// TwinCAT 3 PLC project PLC
// ProgramVersion: 3.1.4026.26
// libraries:
//   Tc2_Standard, * (Beckhoff Automation GmbH)
//   Tc2_System, * (Beckhoff Automation GmbH)
//   Tc2_Utilities, * (Beckhoff Automation GmbH)
//   Tc3_Database, * (Beckhoff Automation GmbH)
//   Tc3_EventLogger, * (Beckhoff Automation GmbH)
// project tree:
//   10_Generator/DUTs/ ST_GeneratorHmi.TcDUT
//   10_Generator/ITFs/ I_Generator.TcIO
//   10_Generator/POUs/ FB_Generator.TcPOU
//   20_RoomTemp/DUTs/ E_CoolingControlState.TcDUT, ST_CoolingControlHmi.TcDUT, ST_RoomTempHmi.TcDUT
//   20_RoomTemp/ITFs/ I_RoomTemp.TcIO
//   20_RoomTemp/POUs/ FB_CoolingControl.TcPOU, FB_RoomTemp.TcPOU, FB_RoomTempControl.TcPOU
//   40_Data/DUTs/ ST_Process_1_Measurements.TcDUT
//   40_Data/POUs/ FB_DataLogger.TcPOU, FB_PLC_DB_Mode.TcPOU, FB_SQL_DB_Mode.TcPOU
//   50_Library/Motors/ITFs/DUTs/ ST_ControlWord.TcDUT, ST_StatusWord.TcDUT
//   50_Library/Motors/ITFs/ I_Motor.TcIO
//   50_Library/Motors/POUs/ FB_MotorAbb.TcPOU, FB_MotorAbb_1.TcPOU
//   99_ESIMERKKI/DUTs/ ST_Esimerkki.TcDUT, ST_EsimerkkiHMI.TcDUT
//   99_ESIMERKKI/POUs/ FB_EsimerkkiToiminto.TcPOU
//   DUTs/ PriceItem.TcDUT, ST_Motors.TcDUT
//   GVLs/ GVL.TcGVL, Motors.TcGVL, Safety.TcGVL
//   / PlcTask.TcTTO
//   POUs/10_aika_ennen_meitä/ FB_AIKA.TcPOU (not stored), FB_HINNAN_ARPOMINEN.TcPOU (not stored), FB_RANK_PRICES.TcPOU
//   POUs/ MAIN.TcPOU
// real-time tasks:
//   TASK PlcTask: cycle T#10ms, priority 20, ADS port 350
// I/O:
//   DEVICE Device 1 (EtherCAT), AmsNetId 192.168.0.154.2.1
//     moottori (FECA-01) [ABB FECA-01 EtherCAT adapter]
// variable links:
//   PLC/PLC Instance <-> Device 1 (EtherCAT)/moottori (FECA-01)
//     PlcTask Inputs/Motors.coolingMotor.nSpeedActual <-> TxPDO 6 map/vl velocity actual value
//     PlcTask Inputs/Motors.coolingMotor.wStatusWord <-> TxPDO 6 map/Statusword
//     PlcTask Outputs/Motors.coolingMotor.nSpeedRef <-> RxPDO 6 map/vl target velocity
//     PlcTask Outputs/Motors.coolingMotor.wControlWord <-> RxPDO 6 map/Controlword

CONFIGURATION PLC
    RESOURCE PLC ON TwinCAT3
        TASK PlcTask(INTERVAL := T#10ms, PRIORITY := 20);
        PROGRAM MAIN WITH PlcTask : MAIN;
    END_RESOURCE
END_CONFIGURATION

// ---- 10_Generator/DUTs/ST_GeneratorHmi.TcDUT
TYPE ST_GeneratorHmi :
STRUCT
	bStart			: BOOL;
	bStop			: BOOL;
	bAltaanTaso		: INT;
	nSahkonKulutus	: INT;
END_STRUCT
END_TYPE

// ---- 20_RoomTemp/DUTs/E_CoolingControlState.TcDUT
{attribute 'qualified_only'}
{attribute 'strict'}
{attribute 'to_string'}
TYPE E_CoolingControlState :
(
	Auto := 0,
	Manual := 1,
	Stop	:= 2,
	Error	:= 3
);
END_TYPE

// ---- 20_RoomTemp/DUTs/ST_CoolingControlHmi.TcDUT
TYPE ST_CoolingControlHmi :
STRUCT
	// HMI -> PLC
	sName					: STRING;
	paramRoomTempSet		: REAL; //
	param_P					: REAL;	//--- PID säätimen parametrit hmi:ltä
	param_I					: REAL;	//
	Param_D					: REAL;	//
	
	bAuto					: BOOL; // Automaatti tila hmi:ltä
	nMotorManualSpeed		: INT;	// Manuaaliajon nopeus hmi:ltä
END_STRUCT
END_TYPE

// ---- 20_RoomTemp/DUTs/ST_RoomTempHmi.TcDUT
TYPE ST_RoomTempHmi :
STRUCT
	// PLC -> HMI
	nRoomTemperature		: REAL;
	sName					: STRING;
	
	// HMI -> PLC
	nValue					: INT := 5; // skaalaus HMI:ltä
	
END_STRUCT
END_TYPE

// ---- 40_Data/DUTs/ST_Process_1_Measurements.TcDUT
TYPE ST_Process_1_Measurements :
STRUCT
	//nID:			LINT;
	//tTime:		DATE_AND_TIME;
	sName:			STRING(50);
	fTemperature:	LREAL;
	fPressure:		LREAL;
	fFlowRate:		LREAL;
END_STRUCT
END_TYPE

// ---- 50_Library/Motors/ITFs/DUTs/ST_ControlWord.TcDUT
TYPE ST_ControlWord :
STRUCT
    // Bitti 0-3: Tilakone ohjaus
    SwitchOn            : BIT;  // Bit 0
    EnableVoltage       : BIT;  // Bit 1
    QuickStop           : BIT;  // Bit 2 — 0 = quick stop aktivoitu
    EnableOperation     : BIT;  // Bit 3

    // Bitti 4-6: Operaatiomoodi spesifinen
    OperationMode0      : BIT;  // Bit 4
    OperationMode1      : BIT;  // Bit 5
    OperationMode2      : BIT;  // Bit 6

    // Bitti 7: Vikareset
    FaultReset          : BIT;  // Bit 7 — nouseva reuna resetoi vian

    // Bitti 8: Halt
    Halt                : BIT;  // Bit 8 — 1 = pysäytä

    // Bitti 9-15: Valmistaja spesifinen
    Reserved9           : BIT;
    Reserved10          : BIT;
    Reserved11          : BIT;
    Reserved12          : BIT;
    Reserved13          : BIT;
    Reserved14          : BIT;
    Reserved15          : BIT;
END_STRUCT
END_TYPE

// ---- 50_Library/Motors/ITFs/DUTs/ST_StatusWord.TcDUT
TYPE ST_StatusWord :
STRUCT
    // Bitti 0-7: Tilakone status
    ReadyToSwitchOn     : BIT;  // Bit 0
    SwitchedOn          : BIT;  // Bit 1
    OperationEnabled    : BIT;  // Bit 2
    Fault               : BIT;  // Bit 3
    VoltageEnabled      : BIT;  // Bit 4
    QuickStop           : BIT;  // Bit 5 — 0 = quick stop aktivoitu
    SwitchOnDisabled    : BIT;  // Bit 6
    Warning             : BIT;  // Bit 7

    // Bitti 8-15
    ManufacturerSpec    : BIT;  // Bit 8
    Remote              : BIT;  // Bit 9  — 1 = väylä ohjaa
    TargetReached       : BIT;  // Bit 10 — 1 = tavoite saavutettu
    InternalLimitActive : BIT;  // Bit 11
    OpModeSpecific0     : BIT;  // Bit 12
    OpModeSpecific1     : BIT;  // Bit 13
    Reserved14          : BIT;  // Bit 14
    Reserved15          : BIT;  // Bit 15
END_STRUCT
END_TYPE

// ---- 99_ESIMERKKI/DUTs/ST_Esimerkki.TcDUT
TYPE ST_Esimerkki :
STRUCT
	
	// Tähän structiin kerätään kaikki Esimerkkitoiminnot, jos niitä on useampia. Helpottaa HMI toimintoja.
	
	stEsimerkki_1			: ST_EsimerkkiHMI;
	stEsimerkki_2			: ST_EsimerkkiHMI;
END_STRUCT
END_TYPE

// ---- 99_ESIMERKKI/DUTs/ST_EsimerkkiHMI.TcDUT
TYPE ST_EsimerkkiHMI :
STRUCT
	bTieto1		: BOOL;
	bTieto2		: BOOL;
	nArvo1		: INT;
END_STRUCT
END_TYPE

// ---- DUTs/PriceItem.TcDUT

TYPE PriceItem : 
STRUCT 
	price : REAL;
	index : INT; 
END_STRUCT 
END_TYPE

// ---- DUTs/ST_Motors.TcDUT
TYPE ST_Motors :
STRUCT
	sName			: STRING;
	bAuto			: BOOL;
	bManual			: BOOL;
	bStop			: BOOL;
	bManualFw		: BOOL;
	bManualBw		: BOOL;
	nManualSpeed	: REAL := 20.0;
	bReset			: BOOL;
	
END_STRUCT
END_TYPE

// ---- GVLs/GVL.TcGVL
{attribute 'qualified_only'}
VAR_GLOBAL
	nTime_multiplier:		INT:=1;
	nSeconds:				INT;
	nMinutes:				INT;
	nHours:					INT;
	nCycle:					INT;
	nMontakohalvinta:		INT(1..95):=20;
	nMontakokalleinta:		INT(1..95):=20;
	nHintaRajaPumppaus:		REAL :=3.0;
	nHintaRajaTuotanto:		REAL :=7.0;
	fprice:					REAL;
	
	// DUT:eissa määriteltiin mitä tietoja structit sisältää. Tässä tehdään muuttuja structissa, jossa tieto asuu. yhdistetään HMI:hin
	stEsimerkki				: ST_Esimerkki;
	
	stGenerator				: ST_GeneratorHmi;
	// Laitoin genun GVL:ään -> helppo työntää rajapinnan kautta tietoja esim roomtempille.
	fbGenerator				: FB_Generator;
	
	stRoomTemp				: ST_RoomTempHmi;
	fbRoomtemp				: FB_RoomTemp;
	
	stCoolingControl		: ST_CoolingControlHmi;
	
	fbDataLogger			: FB_DataLogger;
END_VAR

// ---- GVLs/Motors.TcGVL
{attribute 'qualified_only'}
VAR_GLOBAL
	
	stMotors		: ST_Motors;
	
	
	// Motors
    {attribute 'TcLinkTo' := '.wControlWord := TIID^Device 1 (EtherCAT)^moottori (FECA-01)^RxPDO 6 map^Controlword;
                              .wStatusWord 	:= TIID^Device 1 (EtherCAT)^moottori (FECA-01)^TxPDO 6 map^Statusword;
							  .nSpeedRef	:= TIID^Device 1 (EtherCAT)^moottori (FECA-01)^RxPDO 6 map^vl target velocity;
							  .nSpeedActual := TIID^Device 1 (EtherCAT)^moottori (FECA-01)^TxPDO 6 map^vl velocity actual value'}	
	coolingMotor		: FB_MotorAbb;
END_VAR

// ---- GVLs/Safety.TcGVL
{attribute 'qualified_only'}
VAR_GLOBAL
END_VAR

// ---- 10_Generator/ITFs/I_Generator.TcIO
INTERFACE I_Generator

PROPERTY bRunning : BOOL
GET
END_GET
END_PROPERTY

PROPERTY nHeat : REAL
GET
END_GET
SET
END_SET
END_PROPERTY

END_INTERFACE

// ---- 20_RoomTemp/ITFs/I_RoomTemp.TcIO
INTERFACE I_RoomTemp

PROPERTY nRoomTemp : REAL
GET
END_GET
END_PROPERTY

END_INTERFACE

// ---- 50_Library/Motors/ITFs/I_Motor.TcIO
INTERFACE I_Motor

PROPERTY bAuto : BOOL
GET
END_GET
SET
END_SET
END_PROPERTY

PROPERTY bEnable : BOOL
GET
END_GET
SET
END_SET
END_PROPERTY

PROPERTY bRunning : BOOL
GET
END_GET
END_PROPERTY

PROPERTY nSpeed : INT
GET
END_GET
SET
END_SET
END_PROPERTY

END_INTERFACE

// ---- POUs/MAIN.TcPOU
PROGRAM MAIN
VAR
	// ESIMERKKI TOIMINTO
	fbEsimerkkiToiminto		: FB_EsimerkkiToiminto;
	// -------------------
	fbArvonta:				FB_HINNAN_ARPOMINEN;
	fbTime:					FB_AIKA;
	fbRank:					FB_RANK_PRICES;

	


	nTila					: INT;
	nJarvenAlaraja:			BOOL;
END_VAR

fbTime();
fbRank(arrPrices:=fbArvonta.arrPrices);
gvl.fprice:= fbArvonta.arrPrices[fbTime.onIndex];
nTila	:= GVL.fbGenerator.nTila;

//-------- ESIMERKKI ------------------------------
// Alustetaan ensin esimerkkitoiminto, jonka jälkeen kutsutaan itse funktio
fbEsimerkkiToiminto.Init( refHmi	:= GVL.stEsimerkki.stEsimerkki_1 ); // käy vain alustuksessa
fbEsimerkkiToiminto();													// Pyörii joka kerta
//--------------------------------------------------------------------------

//Suoritetaan arvonta vuorokauden vaihteessa
IF gvl.nSeconds =0 AND gvl.nMinutes = 0 AND gvl.nHours = 0 THEN
	fbArvonta();	
END_IF


//Varmistetaan että aikakerroin on välillä 1-100
IF gvl.nTime_multiplier >100 THEN
	gvl.nTime_multiplier:=100;
END_IF
IF gvl.nTime_multiplier <1 THEN
	gvl.nTime_multiplier:=1;
END_IF


//Varmistetaan että ei mennä yli 96
IF gvl.nMontakohalvinta+gvl.nMontakokalleinta > 96 THEN
	gvl.nMontakokalleinta:= 96-gvl.nMontakohalvinta;
END_IF

// Generaattori ja veden määrät
GVL.fbGenerator.Init(		refHmi := GVL.stGenerator);
GVL.fbGenerator.nRank 		:= fbRank.rank[fbTime.onIndex];
GVL.fbGenerator.nArvonta 	:= fbArvonta.arrPrices[fbTime.onIndex];
GVL.fbGenerator();

// Huoneen lämpötilan simulointi
GVL.fbRoomtemp.Init();
GVL.fbRoomtemp();

// Database yhteys
GVL.fbDataLogger();

END_PROGRAM

// ---- 99_ESIMERKKI/POUs/FB_EsimerkkiToiminto.TcPOU
FUNCTION_BLOCK FB_EsimerkkiToiminto

VAR
	// FB:n sisäiset muuttujat alkumerkki _
	_refHmi		: REFERENCE TO ST_EsimerkkiHMI;
	
	// bInit muuttujaa käytetään silloin, kun ohjelma käynnistetään ensimmäistä kertaa, ja se muuttuu FB_Initissä TRUEKSI
	_bInit		: BOOL;
END_VAR


IF _refHmi.bTieto1 THEN
	_refHmi.nArvo1 := _refHmi.nArvo1 + 1;
END_IF

//FB_Init is always available implicitly and it is used primarily for initialization.
//The return value is not evaluated. For a specific influence, you can also declare the
//methods explicitly and provide additional code there with the standard initialization
//code. You can evaluate the return value.
METHOD FB_Init: BOOL
VAR_INPUT
    bInitRetains: BOOL; // TRUE: the retain variables are initialized (reset warm / reset cold)
    bInCopyCode: BOOL;  // TRUE: the instance will be copied to the copy code afterward (online change)   
END_VAR
_bInit := TRUE;
END_METHOD

METHOD Init
VAR_INPUT
	
	// Muuttuja näkyy ulkomaailmaan, sen takia sillä ei ole _ alkua.
	refHmi		: REFERENCE TO ST_EsimerkkiHMI;
END_VAR
// Alustetaan FB:ssä käytettävät muuttuja, nimet yms...

IF _bInit THEN
	// Välitetään GVL:ssä asuva data FB:n käyttöön.
	// REFERENCE on viittaus GVL listassa olevaan muistialueeseeen.
	_refHmi		REF= refHmi;
END_IF

// Katso MAIN osiosta Esimerkin alustus!!!!!
END_METHOD

END_FUNCTION_BLOCK

// ---- POUs/10_aika_ennen_meitä/FB_RANK_PRICES.TcPOU
FUNCTION_BLOCK FB_RANK_PRICES
VAR_INPUT
	arrPrices: 		ARRAY[1..96] OF REAL; // alkuperäiset hinnat
END_VAR
VAR_OUTPUT
	rank: 			ARRAY[1..96] OF INT; // jokaisen i:n sijoitus 1..96
END_VAR
VAR
	i:				INT;
	j: 				INT;
	arrItems: 		ARRAY[1..96] OF PriceItem; 
	temp: 			PriceItem;
END_VAR

// 1. Kopioi hinnat ja indeksit
FOR i := 1 TO 96 DO
	arrItems[i].price := arrPrices[i];
	arrItems[i].index := i; 
END_FOR

// 2. Järjestä nousevaan järjestykseen 
FOR i := 1 TO 95 DO 
	FOR j := i + 1 TO 96 DO
		IF arrItems[j].price < arrItems[i].price THEN
			temp := arrItems[i];
			arrItems[i] := arrItems[j];
			arrItems[j] := temp;
		END_IF
	END_FOR
END_FOR

// 3. Kirjoita rank alkuperäisille indekseille 
FOR i := 1 TO 96 DO
	rank[arrItems[i].index] := i;
END_FOR

END_FUNCTION_BLOCK

// ---- 10_Generator/POUs/FB_Generator.TcPOU
FUNCTION_BLOCK FB_Generator IMPLEMENTS I_Generator

VAR
	_refHmi					: REFERENCE TO ST_GeneratorHmi;
	_bInit					: BOOL;
	bPumpataan:				BOOL;
	bTuotetaan:				BOOL;
	_nTila:					INT;
	_nRank					: INT;
	_nArvonta				: REAL;
	_nHeat					: REAL;
	
	_fAltaanpinta:			REAL;
	fPinnanmuutos:			REAL:=0.0001;
	nAltaanYlaraja:			BOOL;
	nAltaanAlaraja:			BOOL;
	
END_VAR

// asdasd




PoolSimulation();

StateMachine();

GeneratorHeatSimulation();

UpdateHmi();

PROPERTY bRunning : BOOL
GET
bRunning := bPumpataan OR bTuotetaan;
END_GET
END_PROPERTY

PROPERTY fAltaanpinta : REAL
GET
fAltaanpinta := _fAltaanpinta;
END_GET
SET
_fAltaanpinta := fAltaanpinta;
END_SET
END_PROPERTY

//FB_Init is always available implicitly and it is used primarily for initialization.
//The return value is not evaluated. For a specific influence, you can also declare the
//methods explicitly and provide additional code there with the standard initialization
//code. You can evaluate the return value.
METHOD FB_Init: BOOL
VAR_INPUT
    bInitRetains: BOOL; // TRUE: the retain variables are initialized (reset warm / reset cold)
    bInCopyCode: BOOL;  // TRUE: the instance will be copied to the copy code afterward (online change)   
END_VAR
_bInit := TRUE;
END_METHOD

METHOD GeneratorHeatSimulation : REAL
VAR_INPUT
END_VAR

IF bPumpataan  THEN
	_nHeat 		:= 100;
	
ELSIF bTuotetaan THEN
	_nHeat 		:= ( _refHmi.nSahkonKulutus / 350.0 ) * 100;

ELSE
	_nHeat 		:= 0;
	
END_IF
END_METHOD

METHOD Init
VAR_INPUT
	refHmi		: REFERENCE TO ST_GeneratorHmi;
END_VAR
IF _bInit THEN
	
	_refHmi REF= refHmi;
	
	
	_bInit := FALSE;
END_IF
END_METHOD

PROPERTY nArvonta : REAL
GET
nArvonta := _nArvonta;
END_GET
SET
_nArvonta := nArvonta;
END_SET
END_PROPERTY

PROPERTY nHeat : REAL
GET
nHeat := _nHeat;
END_GET
SET
_nHeat := nHeat;
END_SET
END_PROPERTY

PROPERTY nRank : INT
GET
nRank := _nRank;
END_GET
SET
_nRank := nRank;
END_SET
END_PROPERTY

PROPERTY nTila : INT
GET
nTila := _nTila;
END_GET
END_PROPERTY

METHOD INTERNAL PoolSimulation
VAR_INPUT
END_VAR
//Altaan ylä ja alarajojen simulointi
IF _fAltaanpinta >=99 THEN
	nAltaanYlaraja:= TRUE;
	ELSE
	nAltaanYlaraja:= FALSE;	
END_IF

IF _fAltaanpinta <=1 THEN
	nAltaanAlaraja:= TRUE;
	ELSE
	nAltaanAlaraja:= FALSE;	
END_IF
END_METHOD

METHOD INTERNAL StateMachine
VAR_INPUT
END_VAR
IF _refHmi.bStop THEN
	_refHmi.bStart:=FALSE;
	_refHmi.bStop:= FALSE;
	_nTila:=0;
END_IF


CASE _nTila OF
	0:	//- Stop
		bPumpataan:=FALSE;
		bTuotetaan:=False;
		IF _refHmi.bStart THEN
			_nTila:=1;
			_refHmi.bStart:= FALSE;
		END_IF
		
	1:	// 1 - Odotus
		IF _nRank <= gvl.nMontakohalvinta AND _nArvonta <=  gvl.nHintaRajaPumppaus AND _fAltaanpinta <=100 THEN
			_nTila:=2;
		ELSIF _nRank >= 96-gvl.nMontakokalleinta AND _nArvonta >= gvl.nHintaRajaTuotanto AND _fAltaanpinta >=0THEN
			_nTila:=3;
		END_IF

	2:	// 2 - Pumppaus
		IF _nRank <= gvl.nMontakohalvinta AND _fAltaanpinta <=100 THEN
			bPumpataan:= TRUE;
			_fAltaanpinta:= _fAltaanpinta + fPinnanmuutos*gvl.nTime_multiplier;
		ELSE
			bPumpataan:= FALSE;
			_nTila:=1;
		END_IF		

	3:	//3 - Tuotetaan sähköä
		IF _nRank >= 96-gvl.nMontakokalleinta AND _fAltaanpinta >=0 THEN
			bTuotetaan:= TRUE;
			_fAltaanpinta:= _fAltaanpinta - fPinnanmuutos*gvl.nTime_multiplier;
		ELSE
			bTuotetaan:= FALSE;
			_nTila:=1;
		END_IF	


END_CASE
END_METHOD

METHOD INTERNAL UpdateHmi
VAR_INPUT
END_VAR
_refHmi.bAltaanTaso := REAL_TO_INT(fAltaanpinta);
END_METHOD

END_FUNCTION_BLOCK

// ---- 20_RoomTemp/POUs/FB_RoomTemp.TcPOU
FUNCTION_BLOCK FB_RoomTemp

VAR
	_bInit					: BOOL;
	
	// fb:s
	_fbRoomTempControl		: FB_RoomTempControl;
	_fbCoolingControl		: FB_CoolingControl;
	
	//_fbMotorCooling			: FB_MotorAbb;
	
	
END_VAR


_fbRoomTempControl();
_fbCoolingControl();

//_fbMotorCooling();
Motors.coolingMotor();

//FB_Init is always available implicitly and it is used primarily for initialization.
//The return value is not evaluated. For a specific influence, you can also declare the
//methods explicitly and provide additional code there with the standard initialization
//code. You can evaluate the return value.
METHOD FB_Init: BOOL
VAR_INPUT
    bInitRetains: BOOL; // TRUE: the retain variables are initialized (reset warm / reset cold)
    bInCopyCode: BOOL;  // TRUE: the instance will be copied to the copy code afterward (online change)   
END_VAR
_bInit := TRUE;
END_METHOD

METHOD Init : BOOL
VAR_INPUT
END_VAR
IF _bInit THEN
	



_fbRoomTempControl.Init(	refHmi		:= GVL.stRoomTemp,
							sName		:= 'Generaattori huone',
							iGenerator	:= GVL.fbGenerator);

_fbCoolingControl.Init(	refHmi		:= GVL.stCoolingControl,
						sName		:= 'Generaattori huoneen jäähdytys',
						iMotor		:= Motors.coolingMotor,
						iRoomTemp	:= _fbRoomTempControl );


_bInit := FALSE;
END_IF
END_METHOD

END_FUNCTION_BLOCK

// ---- 20_RoomTemp/POUs/FB_RoomTempControl.TcPOU
FUNCTION_BLOCK FB_RoomTempControl IMPLEMENTS I_RoomTemp

VAR
	// Seuraa onko generaattori päällä (tuottaa/varastoi). Tämän perusteella simuloi lämpötilan nousun.
	// Seruaa onko jäähdytys päällä. Tämän perusteella laskee lämpötilaa.
	_refHmi			: REFERENCE TO ST_RoomTempHmi;
	_bInit			: BOOL;
	_nCycleTime		: REAL := 0.01;
	_nRoomTemp		: REAL := 20.0;
	_nHeatingRate	: REAL;
	
	// Interfaces
	_iGenerator		: I_Generator;
	
	
END_VAR


IF _iGenerator.bRunning THEN
	_nHeatingRate := 0.5 * (_iGenerator.nHeat / 100.0) * (_refHmi.nValue / 100.0);
	
	_nRoomTemp := _nRoomTemp + (_nHeatingRate * _nCycleTime);

ELSIF NOT _iGenerator.bRunning AND _nRoomTemp >= 20.0 THEN
	_nRoomTemp := _nRoomTemp - (0.0005 * _nCycleTime);
	
END_IF



UpdateHmi();

//FB_Init is always available implicitly and it is used primarily for initialization.
//The return value is not evaluated. For a specific influence, you can also declare the
//methods explicitly and provide additional code there with the standard initialization
//code. You can evaluate the return value.
METHOD FB_Init: BOOL
VAR_INPUT
    bInitRetains: BOOL; // TRUE: the retain variables are initialized (reset warm / reset cold)
    bInCopyCode: BOOL;  // TRUE: the instance will be copied to the copy code afterward (online change)   
END_VAR
_bInit := TRUE;
END_METHOD

METHOD Init
VAR_INPUT
	refHmi			: REFERENCE TO ST_RoomTempHmi;
	sName			: STRING;
	iGenerator		: I_Generator;
END_VAR
IF _bInit THEN
	
_refHmi 			REF= refHmi;

_refHmi.sName		:= sName;
_iGenerator			:= iGenerator;

_bInit := FALSE;
END_IF
END_METHOD

PROPERTY nRoomTemp : REAL
GET
nRoomTemp := _nRoomTemp;
END_GET
END_PROPERTY

METHOD INTERNAL UpdateHmi
VAR_INPUT
END_VAR


_refHmi.nRoomTemperature := _nRoomTemp;
END_METHOD

END_FUNCTION_BLOCK

// ---- 20_RoomTemp/POUs/FB_CoolingControl.TcPOU
FUNCTION_BLOCK FB_CoolingControl

VAR
	_bInit			: BOOL;
	
	_refHmi			: REFERENCE TO ST_CoolingControlHmi;
	_iMotor			: I_Motor;
	_iRoomTemp		: I_RoomTemp;
	
	eCoolingState	: E_CoolingControlState;
	
	_fbBasicPID		: FB_BasicPID;
	_nPidOut		: LREAL;
	_nPidOutAbs		: LREAL;
END_VAR

// rajapinnan kautta valvotaan huoneen läpmötilaa. keksitään PID yms säädin, joka nostaa tamun tehoja 
// kun lämpötila nousee...

IF _iMotor.bAuto AND _refHmi.bAuto THEN
	eCoolingState := E_CoolingControlState.Auto;
	
ELSIF NOT _iMotor.bAuto THEN
	eCoolingState := E_CoolingControlState.Manual;
	
	
END_IF

StateMachine();

//FB_Init is always available implicitly and it is used primarily for initialization.
//The return value is not evaluated. For a specific influence, you can also declare the
//methods explicitly and provide additional code there with the standard initialization
//code. You can evaluate the return value.
METHOD FB_Init: BOOL
VAR_INPUT
    bInitRetains: BOOL; // TRUE: the retain variables are initialized (reset warm / reset cold)
    bInCopyCode: BOOL;  // TRUE: the instance will be copied to the copy code afterward (online change)   
END_VAR
_bInit := TRUE;
END_METHOD

METHOD Init : BOOL
VAR_INPUT
	
	refHmi			: REFERENCE TO ST_CoolingControlHmi;
	sName			: STRING;
	iMotor			: I_Motor;
	iRoomTemp		: I_RoomTemp;
END_VAR
IF _bInit THEN
	
	_refHmi			REF= refHmi;
	_refHmi.sName	:= sName;
	_iMotor			:= iMotor;
	_iRoomTemp		:= iRoomTemp;





	_bInit := FALSE;
		
END_IF
END_METHOD

METHOD PRIVATE MotorControl
VAR_INPUT
END_VAR
END_METHOD

METHOD PRIVATE StateMachine : BOOL
VAR_INPUT
END_VAR
CASE eCoolingState OF
	
	E_CoolingControlState.Auto:
		IF _iRoomTemp.nRoomTemp > _refHmi.paramRoomTempSet THEN
			
			_fbBasicPID(	fSetpointValue:= REAL_TO_LREAL(_refHmi.paramRoomTempSet), 
							fActualValue:= REAL_TO_LREAL(_iRoomTemp.nRoomTemp), 
							bReset:= 0, 
							fCtrlCycleTime:= 0.01, 
							fKp:= _refHmi.param_P, 
							fTn:= _refHmi.param_I, 
							fTv:= _refHmi.Param_D, 
							fTd:= 0, 
							fCtrlOutput=> _nPidOut, 
							nErrorStatus=> );
							
							_nPidOutAbs := ABS(_nPidOut);
							_iMotor.nSpeed := LREAL_TO_INT( MAX(0.0, MIN(100.0, _nPidOutAbs)));
							
		END_IF
		
		IF _nPidOutAbs > 5 THEN
		_iMotor.bEnable := TRUE;
		END_IF
		
		
	E_CoolingControlState.Manual:
	;
	
	E_CoolingControlState.Stop:
	;
	
	E_CoolingControlState.Error:
	;
	
END_CASE
END_METHOD

END_FUNCTION_BLOCK

// ---- 40_Data/POUs/FB_DataLogger.TcPOU
FUNCTION_BLOCK FB_DataLogger

VAR
	bTestMode:			BOOL;	(* FALSE: PC, TRUE: PLC *)
	uDevState AT%I*:	UINT;

	bInit:			BOOL := TRUE;
	bStop:			BOOL;
	bDB_Operate:	BOOL;
	fbStartDB: 		NT_StartProcess;	// Start database from USB-stick
	fbStopDB: 		NT_StartProcess;	// Stop database from USB-stick
	fbTON_Init:		TON := (PT:=T#10S);
	fbTON_StopDB:	TON := (PT:=T#10S);
	_fbPlcDBMode	: FB_PLC_DB_Mode;
	_fbSqlDBMode	: FB_SQL_DB_Mode;
END_VAR


IF(bInit) THEN
	fbStartDB(
	NETID:= SEL(bTestMode, '157.24.182.82.1.1', ''),
	PATHSTR:= SEL(bTestMode, 'D:\testMariaStart.bat', 'D:\testMariaStartPLC.bat'),
	DIRNAME:= SEL(bTestMode, 'D:\', 'D:\'),
	COMNDLINE:= ,
	START:= TRUE,
	TMOUT:= T#5S,
	BUSY=> ,
	ERR=> ,
	ERRID=> );

	
	bInit	:= SEL(NOT(fbStartDB.BUSY OR fbStartDB.ERR) AND fbTON_Init.Q, bInit, FALSE);
	bDB_Operate	:= NOT(bInit);
	fbTON_Init(IN:=bInit);
END_IF

IF(bStop) THEN
	fbStopDB(
	NETID:= SEL(bTestMode, '157.24.182.82.1.1', ''),
	PATHSTR:= SEL(bTestMode, 'D:\testMariaStop.bat', 'D:\testMariaStopPLC.bat'),
	DIRNAME:= SEL(bTestMode, 'D:\', 'D:\'),
	COMNDLINE:= ,
	START:= TRUE,
	TMOUT:= T#5S,
	BUSY=> ,
	ERR=> ,
	ERRID=> );

	bStop	:= SEL(NOT(fbStopDB.BUSY OR fbStopDB.ERR) AND fbTON_StopDB.Q, bStop, FALSE);
	bDB_Operate	:= FALSE;
	fbTON_StopDB(IN:=bStop);
END_IF

IF(NOT(bInit) AND bDB_Operate) THEN
	_fbPlcDBMode();
	
	_fbSqlDBMode();
END_IF

END_FUNCTION_BLOCK

// ---- 40_Data/POUs/FB_PLC_DB_Mode.TcPOU
FUNCTION_BLOCK FB_PLC_DB_Mode

VAR
	arrDataName:	ARRAY [0..3] OF STRING(50) := ['reactor_name', 'temperature', 'pressure', 'flow_rate'];	// Database header
	stMeas_1:	ST_Process_1_Measurements	:= (sName:='Reactor 1', fTemperature:=0.1, fPressure:=0.2, fFlowRate:=0.3); // Handled values of the process measurements
	
	fbDB_PLC:	FB_PLCDBWriteEvt(sNetID := '157.24.182.82.1.1', tTimeout := T#5S);	
	//fbDB_PLC:	FB_PLCDBWriteEvt(sNetID := '', tTimeout := T#5S);	// For local DB use

	nCntr:			INT;	// Simple variation for "measurements"
	bWriteRequest:	BOOL;	// Trig single write operation
	bDB_WriteDone:	BOOL;

	tcMessage       :  I_TcMessage;	// For Eventlogger development needs

	fbTON_DataSample:	TON := (PT:=T#5S);
	fbTON_DataStorage:	TON := (PT:=T#1M);
	bLoggingActive:	BOOL;	// Manual activation

END_VAR


	// Create 5s/1min write cycle
fbTON_DataSample(IN:=bLoggingActive);
fbTON_DataStorage(IN:=bLoggingActive);

IF(fbTON_DataSample.Q) THEN
	bWriteRequest	:= TRUE;
	fbTON_DataSample(IN:=FALSE);
END_IF
bLoggingActive	:= SEL(fbTON_DataStorage.Q, bLoggingActive, FALSE);

nCntr	:= SEL(nCntr >= 1000, nCntr + 1, 1);

stMeas_1.fTemperature	:= (INT_TO_LREAL(nCntr)/1000) + 75;
stMeas_1.fPressure		:= (INT_TO_LREAL(nCntr)/1000)*1.5 + 4.1;
stMeas_1.fFlowRate		:= (INT_TO_LREAL(nCntr)/1000)*2.75 + 125;

	// Write used structure into DB
IF(bWriteRequest) THEN
	IF fbDB_PLC.WriteStruct(
        hDBID := 1,
        sTableName := 'reactor_logs',
        pRecord := ADR(stMeas_1),
        cbRecord := SIZEOF(stMeas_1),
        pColumnNames := ADR(arrDataName),
        cbColumnNames := SIZEOF(arrDataName)
    )
    THEN
		IF(NOT(fbDB_PLC.bBusy)) THEN
			bWriteRequest 	:= FALSE;
			bDB_WriteDone	:= TRUE;
		ELSIF(fbDB_PLC.bError) THEN
			tcMessage := fbDB_PLC.ipTcResult;
			bWriteRequest	:= FALSE;
			bDB_WriteDone	:= FALSE;
		END_IF
	END_IF
END_IF

END_FUNCTION_BLOCK

// ---- 40_Data/POUs/FB_SQL_DB_Mode.TcPOU
FUNCTION_BLOCK FB_SQL_DB_Mode

VAR
	nCntr:		INT;

	fbMariaConnection:	FB_SQLDatabaseEvt(sNetID:= '157.24.182.82.1.1', tTimeout:= T#5S);	// DB connection handling
	fbSQLCommand:		FB_SQLCommandEvt(sNetID:= '157.24.182.82.1.1', tTimeout:= T#5S);	// DB read/write operations

	bWriteRequest:		BOOL;	// Trig single write operation
	
	bSQLExecute:		BOOL;
	bSQLDone:			BOOL;
	
	sSQLCmd:			STRING(256);	// Actual SQL command structure to write into DB
	sValue:				STRING(256);	// Stored data into DB

	fbTON_DataSample:	TON := (PT:=T#5S);
	fbTON_DataStorage:	TON := (PT:=T#1M);
	
	bLoggingActive:		BOOL;	// Manual activation
END_VAR


	// Create 5s/1min write cycle
fbTON_DataSample(IN:=bLoggingActive);
fbTON_DataStorage(IN:=bLoggingActive);

bWriteRequest	:= SEL(fbTON_DataSample.Q, bWriteRequest, TRUE);
bLoggingActive	:= SEL(fbTON_DataStorage.Q, bLoggingActive, FALSE);

nCntr	:= SEL(nCntr >= 1000, nCntr + 1, 1);

	// Create connection
IF(NOT(fbMariaConnection.bConnected) AND bWriteRequest) THEN
	fbMariaConnection.Connect(1);
END_IF

	// Create SQL command
IF(fbMariaConnection.bConnected AND bWriteRequest) THEN

	sValue	:= REAL_TO_STRING(INT_TO_REAL(nCntr)/100.0 + 70);
	//sSQLCmd	:= 'INSERT INTO process_measurements (timestamp, tag_name, value, unit) VALUES ( $'2026-09-23 11:01:13$', $'TT_01$', 22.2, $'°C$')';
	sSQLCmd	:= CONCAT('INSERT INTO process_measurements (timestamp, tag_name, value, unit) VALUES (NOW(6),$'TT_01$', ', CONCAT(sValue, ', $'°C$')'));

	fbMariaConnection.CreateCmd(ADR(fbSQLCommand));
	bSQLExecute	:= TRUE;
	bWriteRequest	:= FALSE;
	fbTON_DataSample(IN:=FALSE);
END_IF

	// Execute SQL command
IF(bSQLExecute) THEN
	fbSQLCommand.Execute(
		pSQLCmd:= ADR(sSQLCmd),
		cbSQLCmd:= SIZEOF(sSQLCmd));

	IF(NOT(fbSQLCommand.bBusy)) THEN
		bSQLExecute := FALSE;
		bSQLDone := TRUE;
	END_IF
END_IF

	// Release connection
IF(NOT(fbSQLCommand.bBusy) AND fbMariaConnection.bConnected AND NOT(bLoggingActive)) THEN
	fbMariaConnection.Disconnect();
	bWriteRequest	:= FALSE;
END_IF

END_FUNCTION_BLOCK

// ---- 50_Library/Motors/POUs/FB_MotorAbb.TcPOU
FUNCTION_BLOCK FB_MotorAbb IMPLEMENTS I_Motor

VAR
	// I/O
	wControlWord		AT %Q* : WORD;
	wStatusWord			AT %I* : WORD;
	nSpeedRef			AT %Q* : INT;
	nSpeedActual		AT %I* : INT;

	_bInit				: BOOL;
	_refHmi				: REFERENCE TO ST_Motors;
	
	// States
	_eState				: ( Not_ready_to_switch_on, 
							Switch_on_disabled, 
							Ready_to_Switch_on, Switched_on, 
							Operation_enabled, Quick_stop_active, 
							Fault_reaction_active, Fault, 
							Unknown_state);
							
	_eDriveMode			: ( Disabled, Manual, Auto );
	
	_bQuickStop			: BOOL;
	_bEnable			: BOOL;
	_bRun				: BOOL;
	_nSpeed				: REAL;
	_nSpeedCmd			: REAL;
	_bStopping			: BOOL;
	_bAuto				: BOOL;
	_bManual			: BOOL;
	_bManualFw			: BOOL;
	_bManualBw			: BOOL;
	_nManualSpeed		: REAL := 50;
	
	_bRampDown			: BOOL;
	
	_tonStop			: TON;
END_VAR
VAR CONSTANT
	cScale				: REAL := 200.0;	// 1 % = 200 (100 % = 20000, vrt. ACS880 par. 46.01)
	cStopSpeedLimit		: REAL := 2.0;		// [%] tämän alle -> ajo voidaan estää pysäytyksessä
	
	// StatusWord
	SwMask4F				: WORD := 16#004F;	// bitit 0,1,2,3,6     Päällä
	SwMask6F				: WORD := 16#006F;	// bitit 0,1,2,3,5,6
	SwSwitchOnDisabled 		: WORD := 16#0040;
	SwReadyToSwitchOn		: WORD := 16#0021;
	SwSwitchedOn			: WORD := 16#0023;
	SwOperationEnabled		: WORD := 16#0027;
	SwQuickStopActive		: WORD := 16#0007;
	SwFault					: WORD := 16#0004;
	
	// ControlWord
	CwShutDown				: WORD := 16#0006; // 2, 6, 8
	CwSwitchOn				: WORD := 16#0007; // 3
	CwEnableOperation		: WORD := 16#000F; // 4
	CwDisableOperation		: WORD := 16#0007; // 5
	CwQuickStop				: WORD := 16#0002; // 7, 10, 11
END_VAR


// select state


IF    (wStatusWord AND SwMask4F) = SwSwitchOnDisabled	THEN _eState := Switch_on_disabled;
ELSIF (wStatusWord AND SwMask4F) = SwFault				THEN _eState := Fault;
ELSIF (wStatusWord AND SwMask6F) = SwReadyToSwitchOn	THEN _eState := Ready_to_Switch_on;
ELSIF (wStatusWord AND SwMask6F) = SwSwitchedOn			THEN _eState := Switched_on;
ELSIF (wStatusWord AND SwMask6F) = SwOperationEnabled	THEN _eState := Operation_enabled;
ELSIF (wStatusWord AND SwMask6F) = SwQuickStopActive	THEN _eState := Quick_stop_active;
ELSE                                                         _eState := Unknown_state;
END_IF


// Hallittu pysäytys
_bStopping      := (_eState = Operation_enabled) AND NOT _bEnable;
_toNStop(IN := _bStopping, PT := T#3S);
_bRampDown := _bStopping AND (ABS(nSpeedActual) < cStopSpeedLimit) AND NOT _tonStop.Q;
	
DriveMode();

CASE _eState OF
	
	Quick_stop_active:
	;
	
	Fault:
	;

	Switch_on_disabled:
	wControlWord := CwShutDown;
	
	Ready_to_Switch_on:
	wControlWord := CwSwitchOn;
	
	Switched_on:
	IF _bEnable THEN
		wControlWord := CwEnableOperation;
	END_IF
	
	Operation_enabled:
	IF _bQuickStop THEN
		wControlWord := CwQuickStop;
	END_IF
	
	IF _bStopping THEN
	_nSpeedCmd := 0.0;
		IF _bRampDown THEN	
			wControlWord := CwDisableOperation;
		END_IF
	
	ELSE
		CASE _eDriveMode OF
			Disabled:
			_bRun := FALSE;
			_nSpeedCmd := 0.0;
			
			Manual:
				IF _bManualFw XOR _bManualBw THEN
					_bRun 		:= TRUE;
					_nSpeedCmd 	:= _nManualSpeed;
				ELSE
					_bRun := FALSE;
					_nSpeedCmd 	:= 0.0;
				END_IF
				
			Auto:
			_bRun 		:= _bAuto;
			_nSpeedCmd 	:= _nSpeed;
			
		END_CASE
	END_IF
	
	
END_CASE

nSpeedRef := REAL_TO_INT(LIMIT(-100.0, _nSpeed, 100.0) * cScale);

{warning 'Add property implementation'}
PROPERTY bAuto : BOOL
GET
END_GET
SET
END_SET
END_PROPERTY

{warning 'Add property implementation'}
PROPERTY bEnable : BOOL
GET
END_GET
SET
END_SET
END_PROPERTY

{warning 'Add property implementation'}
PROPERTY bRunning : BOOL
GET
END_GET
END_PROPERTY

METHOD INTERNAL DriveMode : BOOL
VAR_INPUT
END_VAR


IF _bAuto AND NOT _bManual THEN
	_eDriveMode := AUTO;

ELSIF _bManual AND NOT _bAuto THEN
	_eDriveMode := MANUAL;

ELSE
	_eDriveMode := DISABLED;
END_IF


_bManualFw := FALSE;
_bManualBw := FALSE;
IF NOT _bAuto AND _refHmi.bManualFw AND NOT _bManualBw THEN
	_bManualFw := TRUE;
END_IF

IF NOT _bAuto AND _refHmi.bManualBw AND NOT _bManualFw THEN
	_bManualBw := TRUE;
END_IF
END_METHOD

{warning 'Add property implementation'}
PROPERTY nSpeed : INT
GET
END_GET
SET
END_SET
END_PROPERTY

METHOD SetSpeed : INT
VAR_INPUT
	nSpeed		: REAL;
END_VAR
END_METHOD

END_FUNCTION_BLOCK

// ---- 50_Library/Motors/POUs/FB_MotorAbb_1.TcPOU
FUNCTION_BLOCK FB_MotorAbb_1

VAR
	// I/O
	wControlWord		AT %Q* : WORD;
	wStatusWord			AT %I* : WORD;
	nSpeedRef			AT %Q* : INT;
	nSpeedActual		AT %I* : INT;

	_bInit				: BOOL;
	_refHmi				: REFERENCE TO ST_Motors;

	// States
	_eState				: ( Not_ready_to_switch_on, Switch_on_disabled, Ready_to_Switch_on, Switched_on, Operation_enabled, Quick_stop_active, Fault_reaction_active, Fault, Unknown_state );
	_eDriveMode			: ( Disabled, Manual, Auto );					// pyydetty ajotapa
	_eActiveMode		: ( Act_Disabled, Act_Manual, Act_Auto );		// käytössä oleva ajotapa

	// Komennot
	_bQuickStop			: BOOL;			// TRUE = pikapysäytys (kytke NC-hätäseisoista: NOT bOk)
	_bEnable			: BOOL;			// Käyttölupa / päävirta (Switch on)
	_bAuto				: BOOL;			// Ajotavan valinta: automaatti
	_bManual			: BOOL;			// Ajotavan valinta: käsi
	_bAutoRun			: BOOL;			// Käyntikäsky automaattiajossa
	_bReset				: BOOL;			// Vikakuittaus
	_fSpeed				: REAL;			// Automaattiajon nopeus [%]
	_fManualSpeed		: REAL := 10.0;	// Käsiajon nopeus [%]
	_fManualMax			: REAL := 20.0;	// Käsiajon nopeusraja [%]
	_bManualFw			: BOOL;
	_bManualBw			: BOOL;

	// Sisäiset
	_bRunRaw			: BOOL;			// Käyntikäsky valitusta lähteestä
	_bRun				: BOOL;			// Lopullinen käyntipyyntö (luvat + inhibit huomioitu)
	_bPowerReq			: BOOL;			// Päävirta pyydetty (Switch on)
	_bRunInhibit		: BOOL;			// Vaatii uuden käynnistyskäskyn (vika / ajotavan vaihto)
	_bModeChangePending	: BOOL;
	_fSpeedCmd			: REAL;			// Nopeusohje valitusta lähteestä [%]
	_fSpeedRef			: REAL;			// Muuttajalle menevä ohje [%]
	_fSpeedActual		: REAL;			// Toteutunut nopeus [%]
	_bStopping			: BOOL;			// Pysäytys käynnissä (ajo päättyy)
	_bStopped			: BOOL;			// Nopeus alle pysähtymisrajan
	_bRampDown			: BOOL;			// Rampitus kesken -> pidä EnableOperation
	_bWaiting			: BOOL;

	_tStopTimeout		: TIME := T#10S;
	_tonStop			: TON;
	_tonWatch			: TON;
	_rtReset			: R_TRIG;
	_tpReset			: TP;
END_VAR
VAR CONSTANT
	cScale				: REAL := 200.0;	// 1 % = 200 (100 % = 20000, vrt. ACS880 par. 46.01)
	cStopSpeedLimit		: REAL := 2.0;		// [%] tämän alle -> ajo voidaan estää pysäytyksessä

	// StatusWord: maskit ja kuviot (CiA 402)
	SwMask4F				: WORD := 16#004F;	// bitit 0,1,2,3,6
	SwMask6F				: WORD := 16#006F;	// bitit 0,1,2,3,5,6
	SwNotReady				: WORD := 16#0000;	// maski 4F
	SwSwitchOnDisabled 		: WORD := 16#0040;	// maski 4F
	SwFaultReaction			: WORD := 16#000F;	// maski 4F
	SwFault					: WORD := 16#0008;	// maski 4F
	SwReadyToSwitchOn		: WORD := 16#0021;	// maski 6F
	SwSwitchedOn			: WORD := 16#0023;	// maski 6F
	SwOperationEnabled		: WORD := 16#0027;	// maski 6F
	SwQuickStopActive		: WORD := 16#0007;	// maski 6F
	SwBitWarning			: WORD := 16#0080;	// bitti 7
	SwBitRemote				: WORD := 16#0200;	// bitti 9

	// ControlWord
	CwDisableVoltage		: WORD := 16#0004;	// 9, 12; EV=0 (QS pidetään 1:ssä)
	CwShutDown				: WORD := 16#0006;	// 2, 6, 8
	CwSwitchOn				: WORD := 16#0007;	// 3
	CwEnableOperation		: WORD := 16#000F;	// 4
	CwDisableOperation		: WORD := 16#0007;	// 5
	CwQuickStop				: WORD := 16#0002;	// 7, 10, 11
	CwBitFaultReset			: WORD := 16#0080;	// 15: bitti 7, nouseva reuna
END_VAR

// ============================================================
// 0. Ajotavan valinta ja käsiajon suunta HMI:ltä
// ============================================================
DriveMode();

// ============================================================
// 1. Tilan valinta bittimaskilla (kuvio verrataan maskattuun statussanaan)
//    Jos asema ei raportoi bittiä 5: maski 6F -> 4F ja kuviot 21/23/27 -> 01/03/07
// ============================================================
IF    (wStatusWord AND SwMask4F) = SwNotReady			THEN _eState := Not_ready_to_switch_on;
ELSIF (wStatusWord AND SwMask4F) = SwSwitchOnDisabled	THEN _eState := Switch_on_disabled;
ELSIF (wStatusWord AND SwMask4F) = SwFaultReaction		THEN _eState := Fault_reaction_active;
ELSIF (wStatusWord AND SwMask4F) = SwFault				THEN _eState := Fault;
ELSIF (wStatusWord AND SwMask6F) = SwReadyToSwitchOn	THEN _eState := Ready_to_Switch_on;
ELSIF (wStatusWord AND SwMask6F) = SwSwitchedOn			THEN _eState := Switched_on;
ELSIF (wStatusWord AND SwMask6F) = SwOperationEnabled	THEN _eState := Operation_enabled;
ELSIF (wStatusWord AND SwMask6F) = SwQuickStopActive	THEN _eState := Quick_stop_active;
ELSE                                                         _eState := Unknown_state;
END_IF

_fSpeedActual := INT_TO_REAL(nSpeedActual) / cScale;

// ============================================================
// 2. Ajotavan vaihto vain pysäytettynä
// ============================================================
CASE _eDriveMode OF
	Disabled:	_bModeChangePending := (_eActiveMode <> Act_Disabled);
	Manual:		_bModeChangePending := (_eActiveMode <> Act_Manual);
	Auto:		_bModeChangePending := (_eActiveMode <> Act_Auto);
END_CASE

IF _bModeChangePending AND (_eState <> Operation_enabled) THEN
	CASE _eDriveMode OF
		Disabled:	_eActiveMode := Act_Disabled;
		Manual:		_eActiveMode := Act_Manual;
		Auto:		_eActiveMode := Act_Auto;
	END_CASE
	_bRunInhibit        := TRUE;		// ei automaattista käynnistystä vaihdon jälkeen
	_bModeChangePending := FALSE;
END_IF

// ============================================================
// 3. Käyntikäsky ja nopeusohje valitusta lähteestä (joka kierroksella)
// ============================================================
CASE _eActiveMode OF
	Act_Auto:
		_bRunRaw   := _bAutoRun;
		_fSpeedCmd := LIMIT(-100.0, _fSpeed, 100.0);			// rajaa 0..100 jos peruutus ei sallittu

	Act_Manual:
		_bRunRaw   := _bManualFw XOR _bManualBw;
		_fSpeedCmd := LIMIT(0.0, _fManualSpeed, _fManualMax);
		IF _bManualBw THEN
			_fSpeedCmd := -_fSpeedCmd;
		END_IF

	ELSE
		_bRunRaw   := FALSE;
		_fSpeedCmd := 0.0;
END_CASE

IF _bModeChangePending THEN
	_bRunRaw := FALSE;						// pysäytä ensin
END_IF

IF _eState = Fault OR _eState = Fault_reaction_active THEN
	_bRunInhibit := TRUE;					// vian jälkeen vaaditaan uusi käynnistyskäsky
END_IF
IF NOT _bRunRaw THEN
	_bRunInhibit := FALSE;
END_IF

_bPowerReq := _bEnable AND NOT _bQuickStop AND (_eActiveMode <> Act_Disabled);
_bRun      := _bPowerReq AND _bRunRaw AND NOT _bRunInhibit;

// ============================================================
// 4. Hallittu pysäytys: ohje 0 -> odota pysähtymistä (tai timeout) -> Disable operation
// ============================================================
_bStopping := (_eState = Operation_enabled) AND _bPowerReq AND NOT _bRun;
_tonStop(IN := _bStopping, PT := _tStopTimeout);
_bStopped  := ABS(_fSpeedActual) < cStopSpeedLimit;
_bRampDown := _bStopping AND NOT _bStopped AND NOT _tonStop.Q;		// rampitus kesken

// Valvonta: pyydetty tila ei toteudu 5 s kuluessa (STO, Local-tila, kenttäväylä...)
_bWaiting := (_bPowerReq AND (_eState = Not_ready_to_switch_on
                           OR _eState = Switch_on_disabled
                           OR _eState = Ready_to_Switch_on))
          OR (_bRun      AND _eState = Switched_on);
_tonWatch(IN := _bWaiting, PT := T#5S);

// ============================================================
// 5. Vikakuittaus: pulssi 200 ms (bitti 7 on ennen sitä 0 -> nouseva reuna)
// ============================================================
_rtReset(CLK := _bReset);
_tpReset(IN := _rtReset.Q AND (_eState = Fault), PT := T#200MS);

// ============================================================
// 6. Ohjaussana tiloittain (oletus joka kierroksella = ei vanhoja arvoja)
// ============================================================
wControlWord := CwDisableVoltage;

CASE _eState OF

	Not_ready_to_switch_on,
	Fault_reaction_active,
	Unknown_state:
		wControlWord := CwDisableVoltage;				// muuttuja hoitaa itse (0, 1, 14)

	Fault:
		IF _tpReset.Q THEN
			wControlWord := CwDisableVoltage OR CwBitFaultReset;	// (15)
		END_IF

	Switch_on_disabled:
		IF _bPowerReq THEN
			wControlWord := CwShutDown;					// (2)
		END_IF

	Ready_to_Switch_on:
		IF _bPowerReq THEN
			wControlWord := CwSwitchOn;					// (3)
		END_IF											// muuten (7) Disable voltage

	Switched_on:
		IF _bPowerReq THEN
			IF _bRun THEN
				wControlWord := CwEnableOperation;		// (4)
			ELSE
				wControlWord := CwSwitchOn;
			END_IF
		ELSIF _bQuickStop THEN
			wControlWord := CwQuickStop;				// (10)
		ELSE
			wControlWord := CwShutDown;					// (6)
		END_IF

	Operation_enabled:
		IF _bPowerReq THEN
			IF _bRun OR _bRampDown THEN
				wControlWord := CwEnableOperation;		// ajo / hallittu pysäytys
			ELSE
				wControlWord := CwDisableOperation;		// (5) pysähtynyt
			END_IF
		ELSIF _bQuickStop THEN
			wControlWord := CwQuickStop;				// (11), ensisijainen
		ELSE
			wControlWord := CwShutDown;					// (8) lupa pois / Disabled-tila
		END_IF

	Quick_stop_active:
		IF _bQuickStop THEN
			wControlWord := CwQuickStop;				// pidä kunnes pysähtynyt
		END_IF											// muuten (12) Disable voltage
END_CASE

// ============================================================
// 7. Nopeusohje joka kierroksella (-100..100 % -> -20000..20000)
// ============================================================
IF _bRun THEN
	_fSpeedRef := _fSpeedCmd;
ELSE
	_fSpeedRef := 0.0;						// pysäytys ramppia pitkin
END_IF
nSpeedRef := REAL_TO_INT(LIMIT(-100.0, _fSpeedRef, 100.0) * cScale);

PROPERTY bAuto : BOOL
GET
bAuto := _bAuto;
END_GET
SET
_bAuto := bAuto;
END_SET
END_PROPERTY

PROPERTY bAutoRun : BOOL
GET
bAutoRun := _bAutoRun;
END_GET
SET
_bAutoRun := bAutoRun;
END_SET
END_PROPERTY

PROPERTY bEnable : BOOL
GET
bEnable := _bEnable;
END_GET
SET
_bEnable := bEnable;
END_SET
END_PROPERTY

PROPERTY bFault : BOOL
GET
bFault := (_eState = Fault) OR (_eState = Fault_reaction_active);
END_GET
END_PROPERTY

PROPERTY bManual : BOOL
GET
bManual := _bManual;
END_GET
SET
_bManual := bManual;
END_SET
END_PROPERTY

PROPERTY bQuickStop : BOOL
SET
_bQuickStop := bQuickStop;
END_SET
END_PROPERTY

PROPERTY bRemote : BOOL
GET
bRemote := (wStatusWord AND SwBitRemote) <> 0;
END_GET
END_PROPERTY

PROPERTY bReset : BOOL
SET
_bReset := bReset;
END_SET
END_PROPERTY

PROPERTY bRunning : BOOL
GET
bRunning := _eState = Operation_enabled;
END_GET
END_PROPERTY

PROPERTY bTimeout : BOOL
GET
bTimeout := _tonWatch.Q;
END_GET
END_PROPERTY

PROPERTY bWarning : BOOL
GET
bWarning := (wStatusWord AND SwBitWarning) <> 0;
END_GET
END_PROPERTY

METHOD INTERNAL DriveMode : BOOL
VAR_INPUT
END_VAR

IF _bAuto AND NOT _bManual THEN
	_eDriveMode := Auto;
ELSIF _bManual AND NOT _bAuto THEN
	_eDriveMode := Manual;
ELSE
	_eDriveMode := Disabled;			// molemmat tai ei kumpaakaan -> pois
END_IF

// Käsiajon suunta HMI:ltä: molemmat painettuna = ei ajoa
_bManualFw := FALSE;
_bManualBw := FALSE;
IF __ISVALIDREF(_refHmi) AND (_eDriveMode = Manual) THEN
	_bManualFw := _refHmi.bManualFw AND NOT _refHmi.bManualBw;
	_bManualBw := _refHmi.bManualBw AND NOT _refHmi.bManualFw;
END_IF

DriveMode := TRUE;
END_METHOD

PROPERTY fManualSpeed : REAL
GET
fManualSpeed := _fManualSpeed;
END_GET
SET
_fManualSpeed := fManualSpeed;
END_SET
END_PROPERTY

PROPERTY fSpeedActual : REAL
GET
fSpeedActual := _fSpeedActual;
END_GET
END_PROPERTY

PROPERTY nActiveMode : INT
GET
nActiveMode := TO_INT(_eActiveMode);
END_GET
END_PROPERTY

PROPERTY nState : INT
GET
nState := TO_INT(_eState);
END_GET
END_PROPERTY

METHOD SetHmi
VAR_IN_OUT
	stHmi		: ST_Motors;
END_VAR
_refHmi REF= stHmi;
END_METHOD

METHOD SetSpeed : INT
VAR_INPUT
	fSpeed		: REAL;		// Automaattiajon nopeus [%]
END_VAR
_fSpeed := fSpeed;
SetSpeed := REAL_TO_INT(LIMIT(-100.0, fSpeed, 100.0) * cScale);
END_METHOD

END_FUNCTION_BLOCK
